// TIA Portal V16 export
// export: Created 2021-07-12T14:47:19.0493856Z, ExportSetting WithDefaults, DisplayName Totally Integrated Automation Portal, DisplayVersion V16, DisplayName TIA Portal Version Control Interface, DisplayVersion V16, DisplayName TIA Portal Openness, DisplayVersion V16, DisplayName STEP 7 Professional, DisplayVersion V16, DisplayName STEP 7 Safety, DisplayVersion V16, DisplayName WinCC Professional, DisplayVersion V16
TYPE "LSimaHydTO_typeErrorDetail"
TITLE = LSimaHydTO_typeErrorDetail
// Error Details
// stored: IsFailsafeCompliant false
   STRUCT
      Number : UDInt;   // Alarm number
      Reaction : DInt;   // Effective alarm reaction
   END_STRUCT;
END_TYPE
